Staubli VAL3: get.pgx

public program get(string& x_sItem[], num x_nIndex)
  local string l_sKey
  local num i
begin
  // OUTPUT
  // start from the first
  l_sKey=first(saveInOut:cCount)
  // search it
  while l_sKey!=""
    x_sItem=l_sKey
    l_sKey=next(saveInOut:cCount[l_sKey])
    if i==x_nIndex
      return
    else
      i=i+1
    endIf
  endWhile
  // start from the first
  l_sKey=first(saveInOut:aCount)
  while l_sKey!=""
    x_sItem=l_sKey
    l_sKey=next(saveInOut:aCount[l_sKey])
    if i==x_nIndex
      return
    else
      i=i+1
    endIf
  endWhile
end
